{attribute 'qualified_only'}
{attribute 'to_string'}
TYPE CornerGuard :
(
	COR48 := 1,
	COR96,
	
	size
);
END_TYPE

(* stored: Version 1.1.0.1, ProductVersion 3.1.4024.11
   DUT CornerGuard: Id {99dc40db-6ff9-4ed3-9f8b-8510d0804786} *)
